{attribute 'GeneratedUsingTerminal: EL2212-0000-0020'}
{attribute addProperty BoxType "EL2212-0000-0020"}
{attribute addProperty Description "EL2212 2Ch. dig. output with overexcitation (24V DC, 2.5A, 10A Peak)"}
{attribute addProperty Physics "KK"}
{attribute addProperty Id "DOX_Status_Channel_1AT %I*DOX_Status_Channel_6FDDBA987DOX_Status_Channel_2AT %I*DOX_Status_Channel_6FDDBA987DOX_Control_Channel_1AT %Q*DOX_Control_Channel_E69306414DOX_Control_Channel_2AT %Q*DOX_Control_Channel_E69306414WcStateAT %I*WcState_9091E0EB2InfoDataAT %I*InfoData_32EB74EA10"}
{attribute addProperty CRC "3336464230"}
{attribute addProperty Size "34"}
TYPE EL2212_C6DE6766 EXTENDS EtcSlaveTerminalBase_947E5A46 :
STRUCT
	{attribute addProperty Name "DOX_Status_Channel_1"}
	DOX_Status_Channel_1 : DOX_Status_Channel_6FDDBA98;
	{attribute addProperty Name "DOX_Status_Channel_2"}
	DOX_Status_Channel_2 : DOX_Status_Channel_6FDDBA98;
	{attribute addProperty Name "DOX_Control_Channel_1"}
	DOX_Control_Channel_1 : DOX_Control_Channel_E6930641;
	{attribute addProperty Name "DOX_Control_Channel_2"}
	DOX_Control_Channel_2 : DOX_Control_Channel_E6930641;
	{attribute addProperty Name "WcState"}
	WcState : WcState_9091E0EB;
	{attribute addProperty Name "InfoData"}
	InfoData : InfoData_32EB74EA;
END_STRUCT
END_TYPE

(* stored: Version 1.2.0.0, ProductVersion 3.1.4024.11
   DUT EL2212_C6DE6766: Id {8efe4069-c4f1-4f5b-ab0c-32e4dc6bc756} *)
